TYPE "ProcessCheck_ShW"
VERSION : 0.1
   STRUCT
      Trigger : Bool;
      Mode : String[48];
      Result : Int;
      Completed : Bool;
   END_STRUCT;

END_TYPE

